FUNCTION AlarmParametersProvider : AlarmParameters
VAR_INPUT
	CurrentParameterValue : REAL;
	MaxParameterLimit : REAL;
	MinParameterLimit : REAL;
END_VAR
VAR
	alarmParameters : AlarmParameters;
END_VAR

alarmParameters.CurrentParameterValue := CurrentParameterValue;
alarmParameters.MaxParameterLimit := MaxParameterLimit;
alarmParameters.MinParameterLimit := MinParameterLimit;

AlarmParametersProvider := alarmParameters;

END_FUNCTION

(* stored: Version 1.1.0.1, ProductVersion 3.1.4022.16
   POU AlarmParametersProvider: Id {8ba4abda-c032-4f0e-b698-86b788877820}, SpecialFunc None *)
